FUNCTION_BLOCK SELECT_ACTIVE_FEEDER_SEQ
VAR_INPUT
END_VAR
VAR_OUTPUT
END_VAR
VAR
END_VAR

END_FUNCTION_BLOCK

(* stored: Version 1.1.0.1, ProductVersion 3.1.4022.18
   POU SELECT_ACTIVE_FEEDER_SEQ: Id {c85cf2b2-f7f2-4ead-a0b3-57d755304991}, SpecialFunc None *)
